(* Logix 5000 project; controller GEA_Test_Chamber vendor 1 type 14 code 196 rev 32.14; software revision 32.04; part 3 of 11 *)
(* tags used below, declared in another part *)
   Inp_Enable : BOOL;
   Ref_Connection : raC_UDT_ModbusServerBase;
   Ref_ModbusData : raC_UDT_ModbusServerData;
   Sts_ActiveConnections : DINT;   // Number of currently active Client connections.
   Ref_MsgDelete : MESSAGE;
   Ref_MsgDeleteAll : MESSAGE;
   Sts_EN : BOOL;
   Sts_Waiting : BOOL;
   Sts_Accepted : BOOL;
   Sts_Faulted : BOOL;
   Sts_LastError : DINT;   // The last recorded socket error for this connection. 0 good, -2- Write Error, -4 - Read Error, -6 connection failed, -7 D
   Wrk_MSGStep : DINT;
   Wrk_BaseInstance : DINT;
   Wrk_WrIndex : DINT;
   Wrk_TransIndex : DINT;
   Wrk_TimerIndex : DINT;
   Wrk_ClrReqIndex : DINT;
   Wrk_AcceptInstance : DINT;
   Wrk_InstSize : DINT;
   Wrk_RdWrIndex : DINT;
   Wrk_TempActConn : DINT;
   Wrk_InstIndex : DINT;
   Wrk_LastInstIndex : DINT;
   Wrk_OkToIncement : BOOL;
   Wrk_StepLockTimer : TIMER;
   Wrk_TempTime : DINT;
   Wrk_Instances : raC_UDT_ModbusServerRWSocket[10];
   Wrk_Controller_Type : DINT;
   Wrk_Controller_Name : SINT[33];
   Wrk_InitCompleted : BOOL;
   Wrk_InstIndex2 : DINT;
   Wrk_InstIndex3 : DINT;
   HMI_Tab : DINT;
   wrk_temp_Instances : raC_UDT_ModbusServerRWSocketInfo[10];
   wrk_FAL_Addr : CONTROL;
   wrk_LoopIndex : DINT;
   wrk_AddrIndex : DINT;
   HMI : raC_UDT_ModbusServerHMI;
   wrk_FAL_01 : CONTROL;
(* raC_Opr_NetModbusTCPServer, continued *)

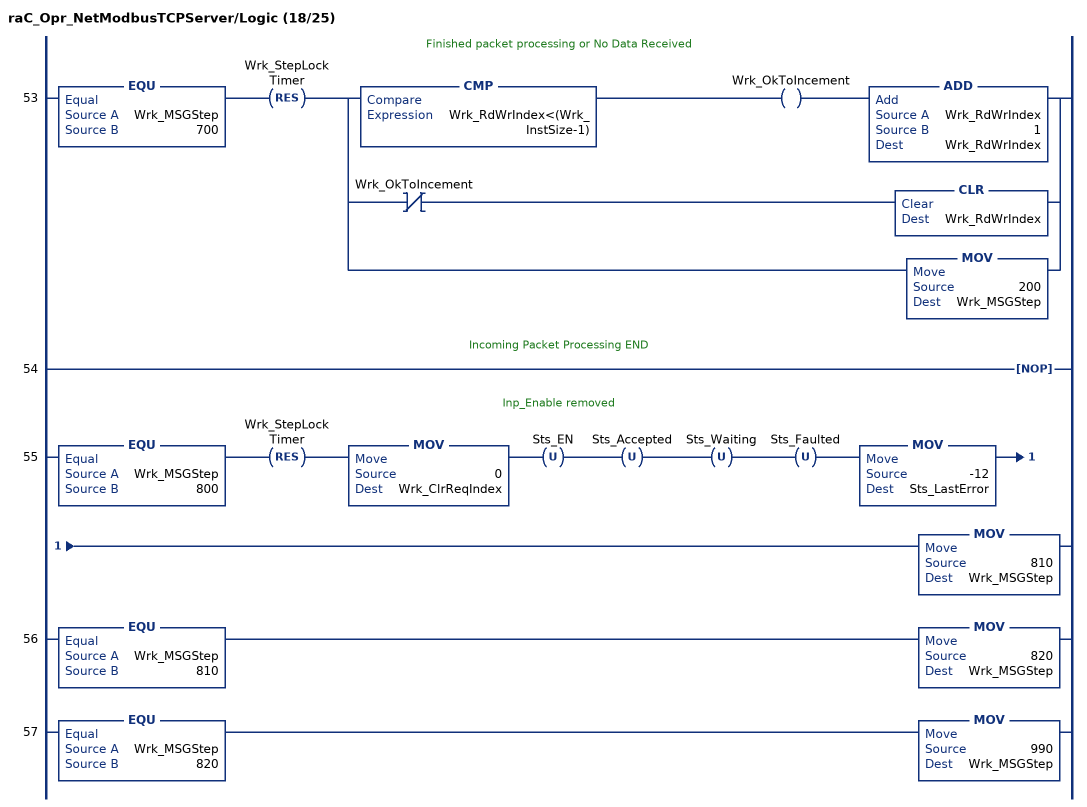
   // Finished packet processing or No Data Received
   53: EQU(Wrk_MSGStep,700)RES(Wrk_StepLockTimer)[CMP(Wrk_RdWrIndex<(Wrk_InstSize-1)) OTE(Wrk_OkToIncement) ADD(Wrk_RdWrIndex,1,Wrk_RdWrIndex) ,XIO(Wrk_OkToIncement) CLR(Wrk_RdWrIndex) ,MOV(200,Wrk_MSGStep) ];
   // Incoming Packet Processing END
   54: NOP();
   // Inp_Enable removed
   55: EQU(Wrk_MSGStep,800)RES(Wrk_StepLockTimer)MOV(0,Wrk_ClrReqIndex)OTU(Sts_EN)OTU(Sts_Accepted)OTU(Sts_Waiting)OTU(Sts_Faulted)MOV(-12,Sts_LastError)MOV(810,Wrk_MSGStep);
   56: EQU(Wrk_MSGStep,810)MOV(820,Wrk_MSGStep);
   57: EQU(Wrk_MSGStep,820)MOV(990,Wrk_MSGStep);
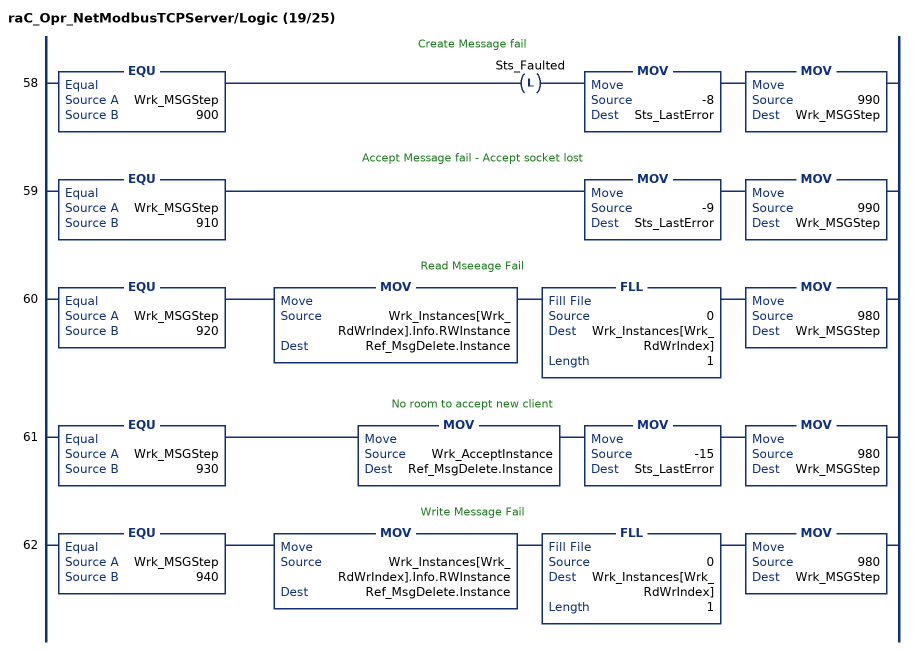
   // Create Message fail
   58: EQU(Wrk_MSGStep,900)OTL(Sts_Faulted)MOV(-8,Sts_LastError)MOV(990,Wrk_MSGStep);
   // Accept Message fail - Accept socket lost
   59: EQU(Wrk_MSGStep,910)MOV(-9,Sts_LastError)MOV(990,Wrk_MSGStep);
   // Read Mseeage Fail
   60: EQU(Wrk_MSGStep,920)MOV(Wrk_Instances[Wrk_RdWrIndex].Info.RWInstance,Ref_MsgDelete.Instance)FLL(0,Wrk_Instances[Wrk_RdWrIndex],1)MOV(980,Wrk_MSGStep);
   // No room to accept new client
   61: EQU(Wrk_MSGStep,930)MOV(Wrk_AcceptInstance,Ref_MsgDelete.Instance)MOV(-15,Sts_LastError)MOV(980,Wrk_MSGStep);
   // Write Message Fail
   62: EQU(Wrk_MSGStep,940)MOV(Wrk_Instances[Wrk_RdWrIndex].Info.RWInstance,Ref_MsgDelete.Instance)FLL(0,Wrk_Instances[Wrk_RdWrIndex],1)MOV(980,Wrk_MSGStep);
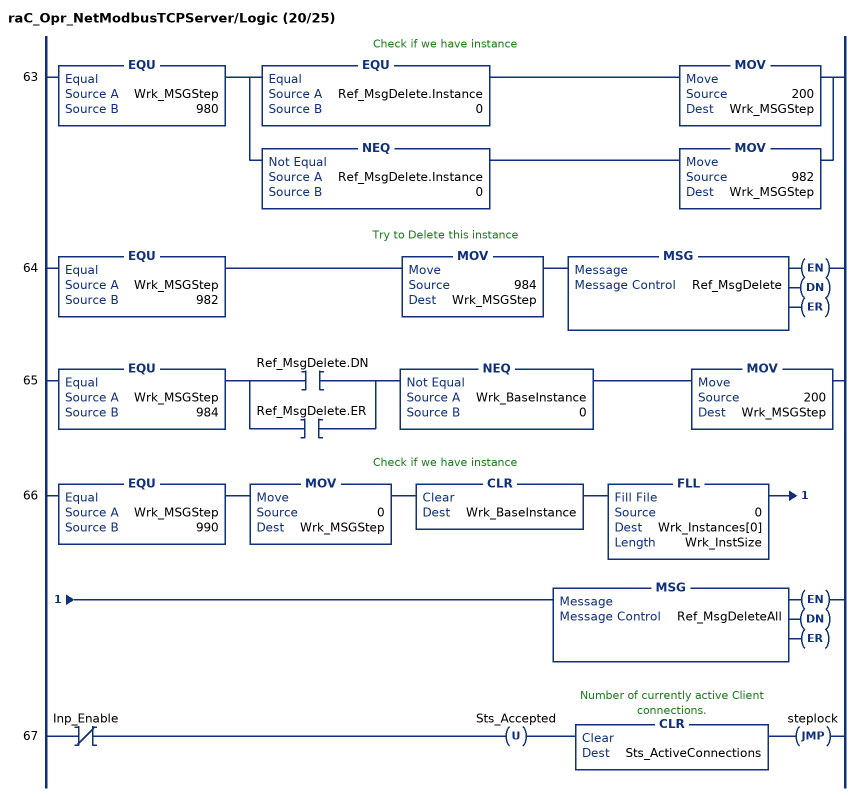
   // Check if we have instance
   63: EQU(Wrk_MSGStep,980)[EQU(Ref_MsgDelete.Instance,0) MOV(200,Wrk_MSGStep) ,NEQ(Ref_MsgDelete.Instance,0) MOV(982,Wrk_MSGStep) ];
   // Try to Delete this instance
   64: EQU(Wrk_MSGStep,982)MOV(984,Wrk_MSGStep)MSG(Ref_MsgDelete);
   65: EQU(Wrk_MSGStep,984)[XIC(Ref_MsgDelete.DN) ,XIC(Ref_MsgDelete.ER) ]NEQ(Wrk_BaseInstance,0)MOV(200,Wrk_MSGStep);
   // Check if we have instance
   66: EQU(Wrk_MSGStep,990)MOV(0,Wrk_MSGStep)CLR(Wrk_BaseInstance)FLL(0,Wrk_Instances[0],Wrk_InstSize)MSG(Ref_MsgDeleteAll);
   67: XIO(Inp_Enable)OTU(Sts_Accepted)CLR(Sts_ActiveConnections)JMP(steplock);
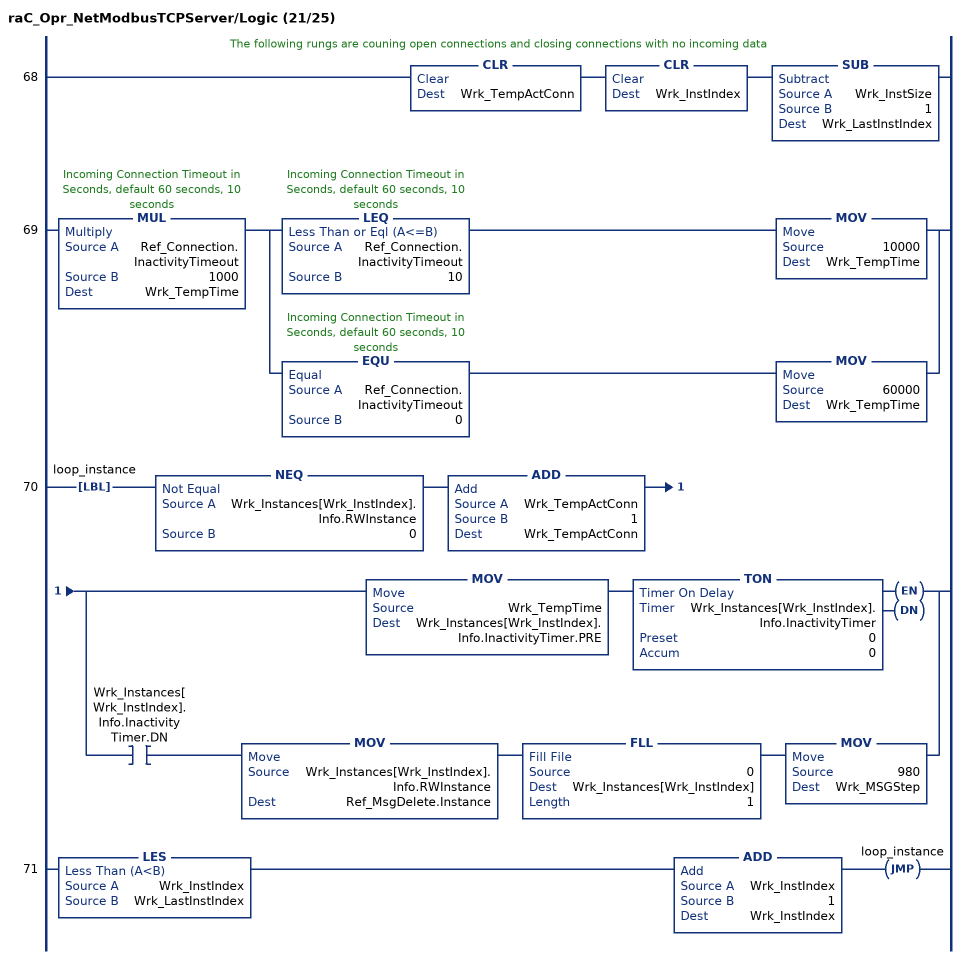
   // The following rungs are couning open connections and closing connections with no incoming data
   68: CLR(Wrk_TempActConn)CLR(Wrk_InstIndex)SUB(Wrk_InstSize,1,Wrk_LastInstIndex);
   69: MUL(Ref_Connection.InactivityTimeout,1000,Wrk_TempTime)[LEQ(Ref_Connection.InactivityTimeout,10) MOV(10000,Wrk_TempTime) ,EQU(Ref_Connection.InactivityTimeout,0) MOV(60000,Wrk_TempTime) ];
   70: LBL(loop_instance)NEQ(Wrk_Instances[Wrk_InstIndex].Info.RWInstance,0)ADD(Wrk_TempActConn,1,Wrk_TempActConn)[MOV(Wrk_TempTime,Wrk_Instances[Wrk_InstIndex].Info.InactivityTimer.PRE) TON(Wrk_Instances[Wrk_InstIndex].Info.InactivityTimer,0,0) ,XIC(Wrk_Instances[Wrk_InstIndex].Info.InactivityTimer.DN) MOV(Wrk_Instances[Wrk_InstIndex].Info.RWInstance,Ref_MsgDelete.Instance) FLL(0,Wrk_Instances[Wrk_InstIndex],1) MOV(980,Wrk_MSGStep) ];
   71: LES(Wrk_InstIndex,Wrk_LastInstIndex)ADD(Wrk_InstIndex,1,Wrk_InstIndex)JMP(loop_instance);
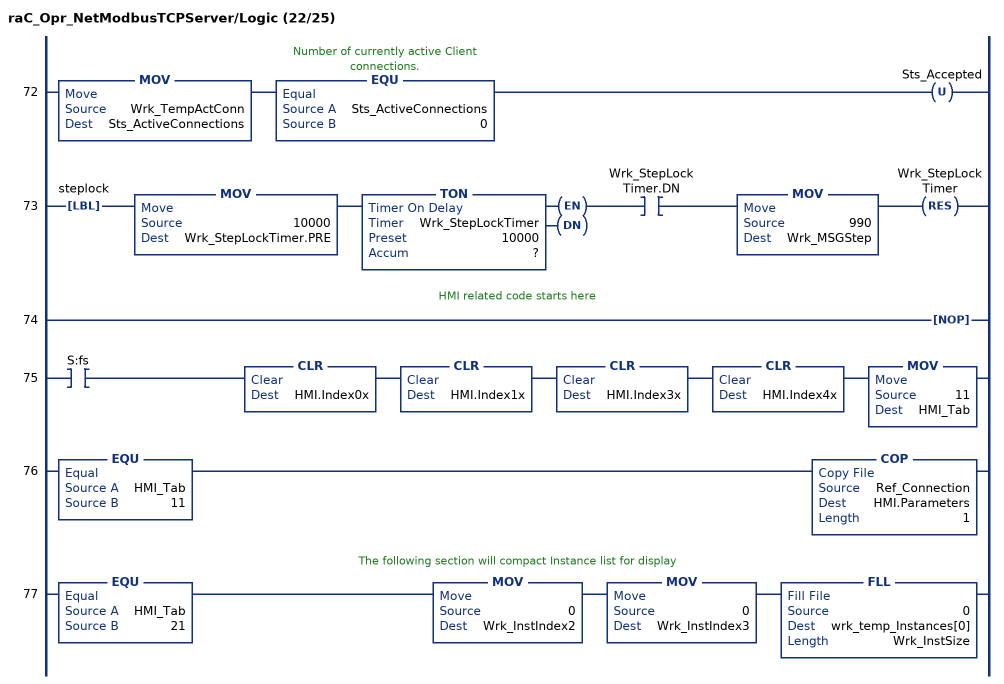
   72: MOV(Wrk_TempActConn,Sts_ActiveConnections)EQU(Sts_ActiveConnections,0)OTU(Sts_Accepted);
   73: LBL(steplock)MOV(10000,Wrk_StepLockTimer.PRE)TON(Wrk_StepLockTimer,?,?)XIC(Wrk_StepLockTimer.DN)MOV(990,Wrk_MSGStep)RES(Wrk_StepLockTimer);
   // HMI related code starts here
   74: NOP();
   75: XIC(S:fs)CLR(HMI.Index0x)CLR(HMI.Index1x)CLR(HMI.Index3x)CLR(HMI.Index4x)MOV(11,HMI_Tab);
   76: EQU(HMI_Tab,11)COP(Ref_Connection,HMI.Parameters,1);
   // The following section will compact Instance list for display
   77: EQU(HMI_Tab,21)MOV(0,Wrk_InstIndex2)MOV(0,Wrk_InstIndex3)FLL(0,wrk_temp_Instances[0],Wrk_InstSize);
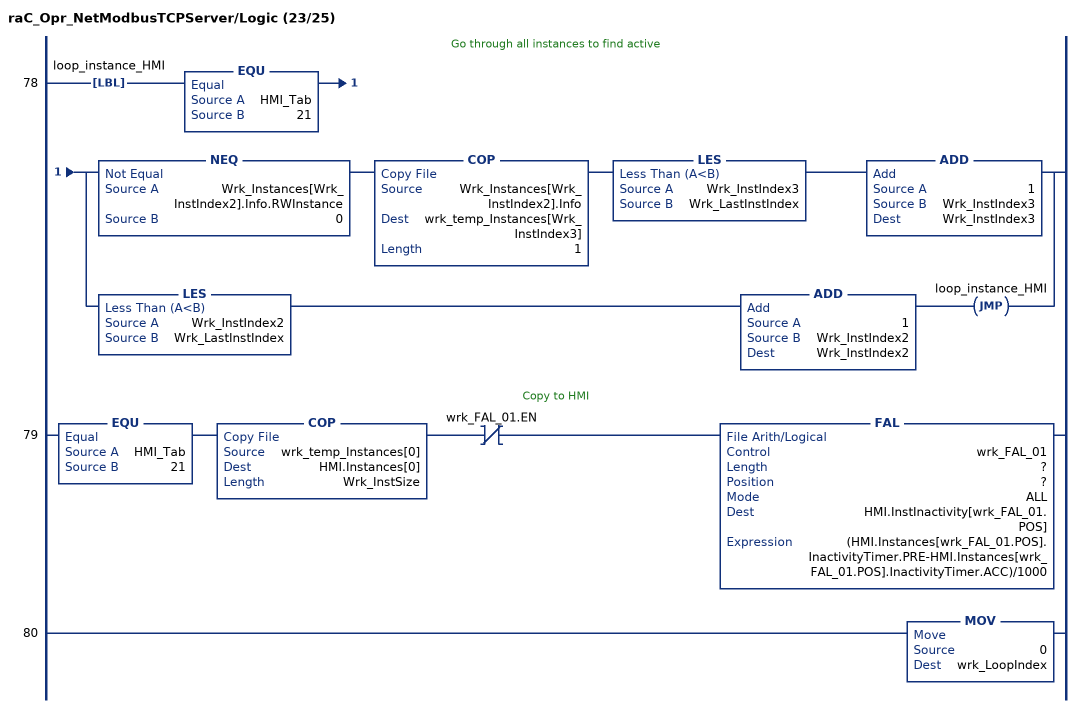
   // Go through all instances to find active
   78: LBL(loop_instance_HMI)EQU(HMI_Tab,21)[NEQ(Wrk_Instances[Wrk_InstIndex2].Info.RWInstance,0) COP(Wrk_Instances[Wrk_InstIndex2].Info,wrk_temp_Instances[Wrk_InstIndex3],1) LES(Wrk_InstIndex3,Wrk_LastInstIndex) ADD(1,Wrk_InstIndex3,Wrk_InstIndex3) ,LES(Wrk_InstIndex2,Wrk_LastInstIndex) ADD(1,Wrk_InstIndex2,Wrk_InstIndex2) JMP(loop_instance_HMI) ];
   // Copy to HMI
   79: EQU(HMI_Tab,21)COP(wrk_temp_Instances[0],HMI.Instances[0],Wrk_InstSize)XIO(wrk_FAL_01.EN)FAL(wrk_FAL_01,?,?,ALL,HMI.InstInactivity[wrk_FAL_01.POS],(HMI.Instances[wrk_FAL_01.POS].InactivityTimer.PRE-HMI.Instances[wrk_FAL_01.POS].InactivityTimer.ACC)/1000);
   80: MOV(0,wrk_LoopIndex);
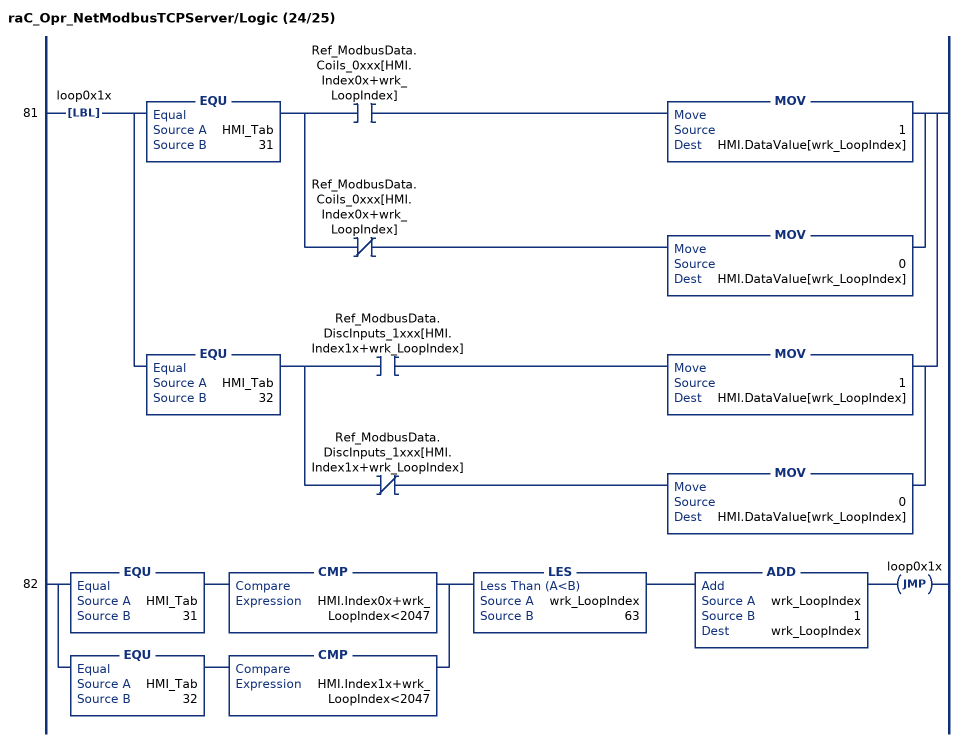
   81: LBL(loop0x1x)[EQU(HMI_Tab,31) [XIC(Ref_ModbusData.Coils_0xxx[HMI.Index0x+wrk_LoopIndex]) MOV(1,HMI.DataValue[wrk_LoopIndex]) ,XIO(Ref_ModbusData.Coils_0xxx[HMI.Index0x+wrk_LoopIndex]) MOV(0,HMI.DataValue[wrk_LoopIndex]) ] ,EQU(HMI_Tab,32) [XIC(Ref_ModbusData.DiscInputs_1xxx[HMI.Index1x+wrk_LoopIndex]) MOV(1,HMI.DataValue[wrk_LoopIndex]) ,XIO(Ref_ModbusData.DiscInputs_1xxx[HMI.Index1x+wrk_LoopIndex]) MOV(0,HMI.DataValue[wrk_LoopIndex]) ] ];
   82: [EQU(HMI_Tab,31) CMP(HMI.Index0x+wrk_LoopIndex<2047) ,EQU(HMI_Tab,32) CMP(HMI.Index1x+wrk_LoopIndex<2047) ]LES(wrk_LoopIndex,63)ADD(wrk_LoopIndex,1,wrk_LoopIndex)JMP(loop0x1x);
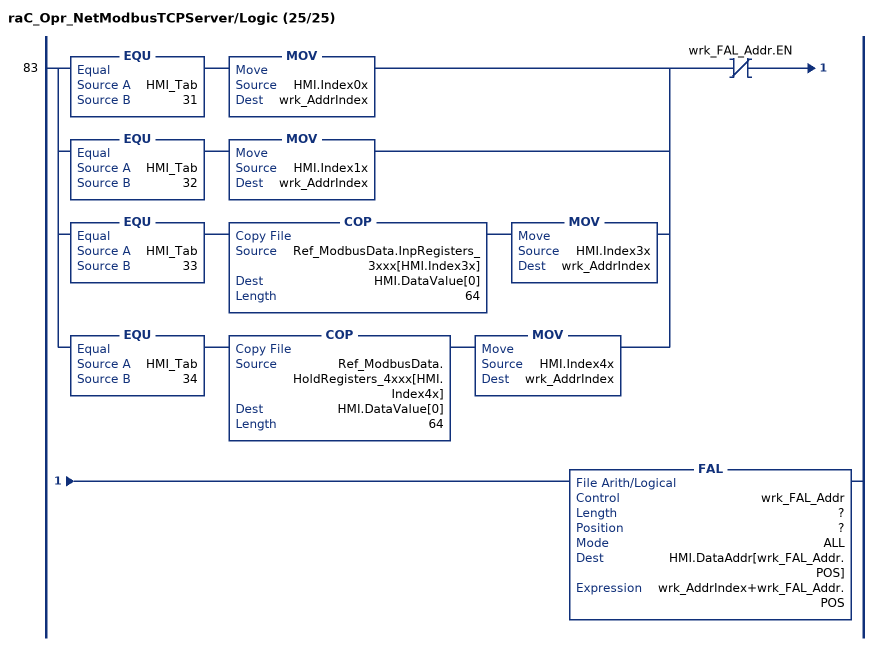
   83: [EQU(HMI_Tab,31) MOV(HMI.Index0x,wrk_AddrIndex) ,EQU(HMI_Tab,32) MOV(HMI.Index1x,wrk_AddrIndex) ,EQU(HMI_Tab,33) COP(Ref_ModbusData.InpRegisters_3xxx[HMI.Index3x],HMI.DataValue[0],64) MOV(HMI.Index3x,wrk_AddrIndex) ,EQU(HMI_Tab,34) COP(Ref_ModbusData.HoldRegisters_4xxx[HMI.Index4x],HMI.DataValue[0],64) MOV(HMI.Index4x,wrk_AddrIndex) ]XIO(wrk_FAL_Addr.EN)FAL(wrk_FAL_Addr,?,?,ALL,HMI.DataAddr[wrk_FAL_Addr.POS],wrk_AddrIndex+wrk_FAL_Addr.POS);
END_ROUTINE

ROUTINE Prescan   (* ladder *)
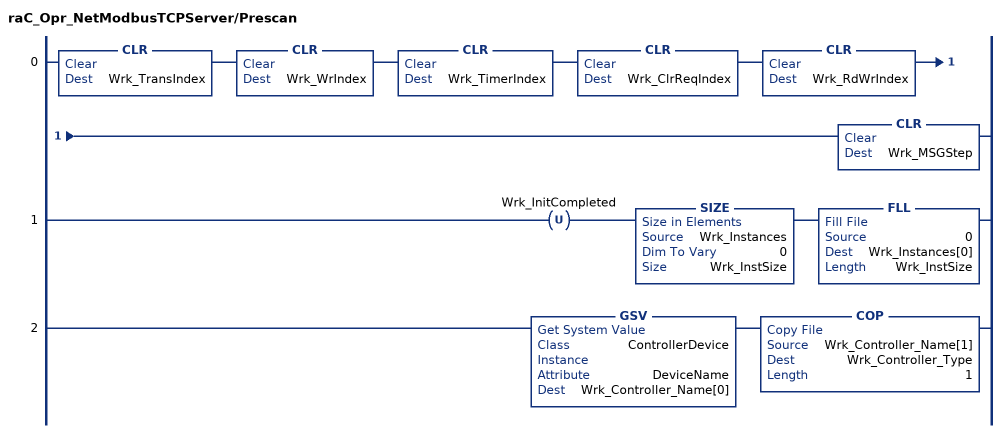
   0: CLR(Wrk_TransIndex)CLR(Wrk_WrIndex)CLR(Wrk_TimerIndex)CLR(Wrk_ClrReqIndex)CLR(Wrk_RdWrIndex)CLR(Wrk_MSGStep);
   1: OTU(Wrk_InitCompleted)SIZE(Wrk_Instances,0,Wrk_InstSize)FLL(0,Wrk_Instances[0],Wrk_InstSize);
   2: GSV(ControllerDevice,,DeviceName,Wrk_Controller_Name[0])COP(Wrk_Controller_Name[1],Wrk_Controller_Type,1);
END_ROUTINE
END_ADD_ON_INSTRUCTION

ADD_ON_INSTRUCTION raC_Tec_NetModbusTCPClient_BuildReqStr   (* revision 2.1, ExecutePrescan *)
// This routine builds a request string.
// Revision note:
// Moved to DINT in BeginAddress with boundary enforcement
VAR_IN_OUT
   Transaction : raC_UDT_ModbusClientTransaction; {required}
   ModbusData : raC_UDT_ModbusClientData; {required}
END_VAR
VAR_OUTPUT
   ER : BOOL; {access Read Only, visible}
END_VAR
VAR
   Wrk_TempInt : INT; {access None}
   Wrk_TempBeginInt : INT; {access None}
   Wrk_TempASCII_462 : STR0462; {access None}
   Wrk_Bit : DINT; {access None}
   Wrk_Byte : DINT; {access None}
   Wrk_Index : DINT; {access None}
   Wrk_LastAddr : DINT; {access None}
   Wrk_ValidRemoteRange : BOOL; {access None}
END_VAR

ROUTINE Logic   (* ladder *)
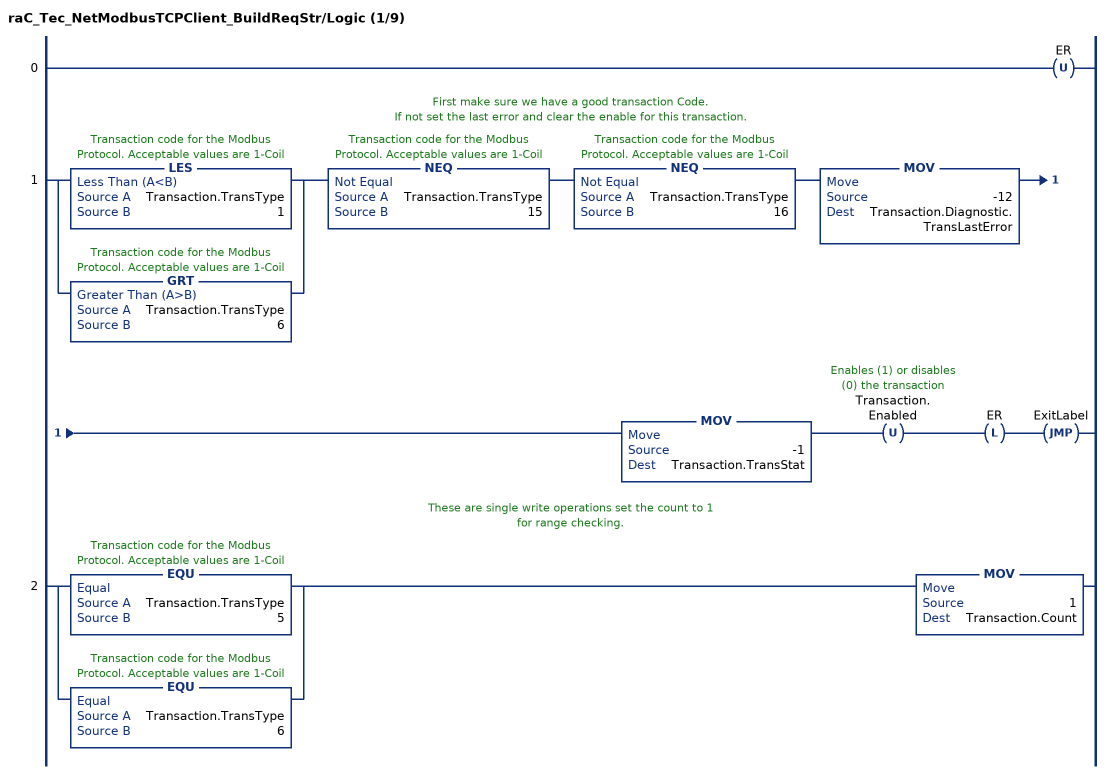
   0: OTU(ER);
   // First make sure we have a good transaction Code.
   // If not set the last error and clear the enable for this transaction.
   1: [LES(Transaction.TransType,1) ,GRT(Transaction.TransType,6) ]NEQ(Transaction.TransType,15)NEQ(Transaction.TransType,16)MOV(-12,Transaction.Diagnostic.TransLastError)MOV(-1,Transaction.TransStat)OTU(Transaction.Enabled)OTL(ER)JMP(ExitLabel);
   // These are single write operations set the count to 1
   //  for range checking.
   2: [EQU(Transaction.TransType,5) ,EQU(Transaction.TransType,6) ]MOV(1,Transaction.Count);
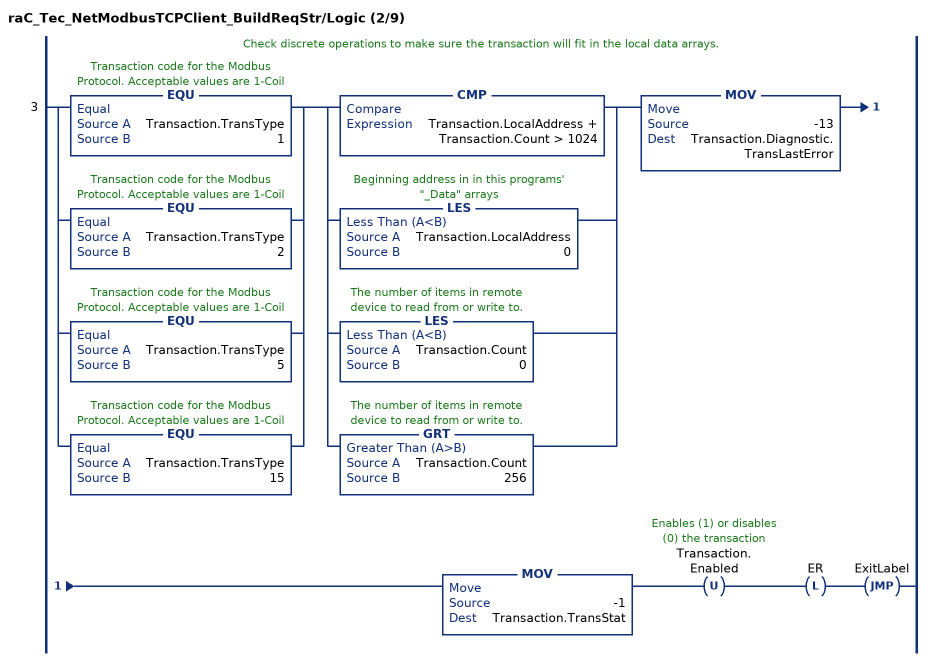
   // Check discrete operations to make sure the transaction will fit in the local data arrays.
   3: [EQU(Transaction.TransType,1) ,EQU(Transaction.TransType,2) ,EQU(Transaction.TransType,5) ,EQU(Transaction.TransType,15) ][CMP(Transaction.LocalAddress + Transaction.Count > 1024) ,LES(Transaction.LocalAddress,0) ,LES(Transaction.Count,0) ,GRT(Transaction.Count,256) ]MOV(-13,Transaction.Diagnostic.TransLastError)MOV(-1,Transaction.TransStat)OTU(Transaction.Enabled)OTL(ER)JMP(ExitLabel);
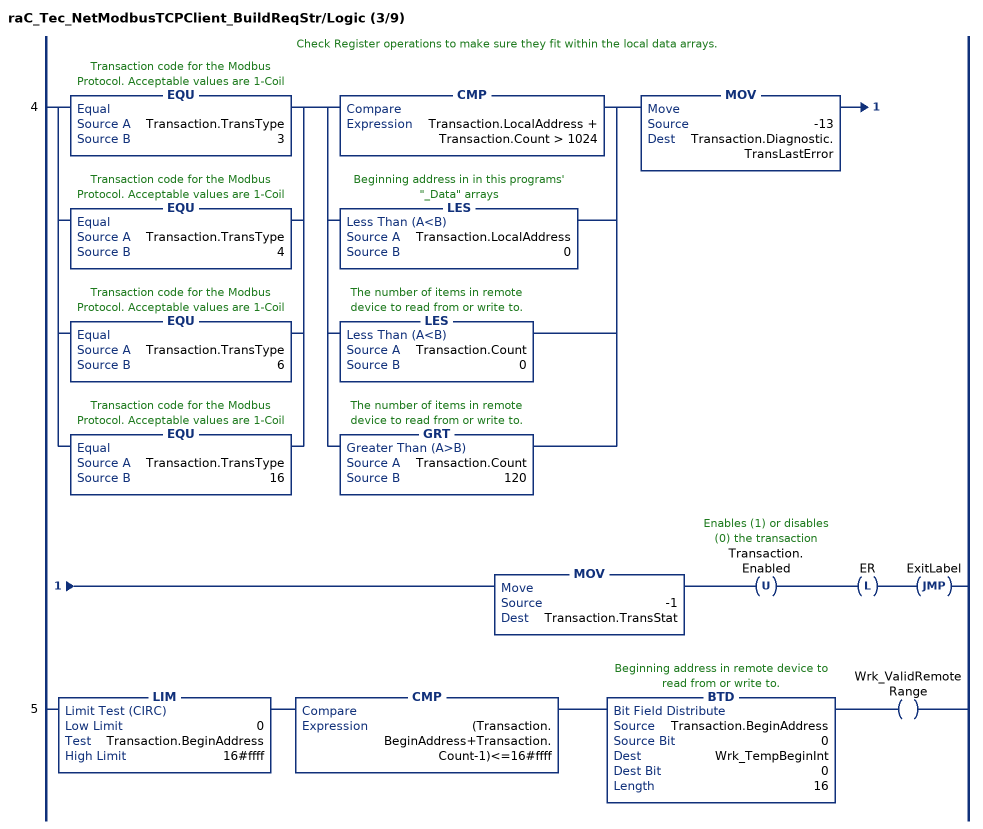
   // Check Register operations to make sure they fit within the local data arrays.
   4: [EQU(Transaction.TransType,3) ,EQU(Transaction.TransType,4) ,EQU(Transaction.TransType,6) ,EQU(Transaction.TransType,16) ][CMP(Transaction.LocalAddress + Transaction.Count > 1024) ,LES(Transaction.LocalAddress,0) ,LES(Transaction.Count,0) ,GRT(Transaction.Count,120) ]MOV(-13,Transaction.Diagnostic.TransLastError)MOV(-1,Transaction.TransStat)OTU(Transaction.Enabled)OTL(ER)JMP(ExitLabel);
   5: LIM(0,Transaction.BeginAddress,16#ffff)CMP((Transaction.BeginAddress+Transaction.Count-1)<=16#ffff)BTD(Transaction.BeginAddress,0,Wrk_TempBeginInt,0,16)OTE(Wrk_ValidRemoteRange);
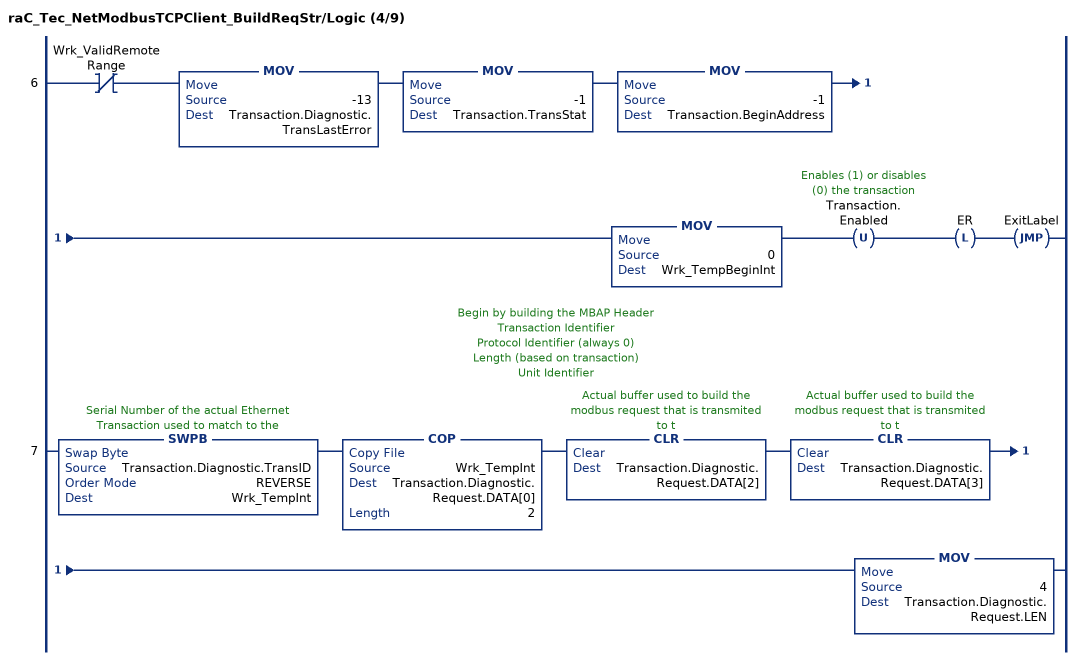
   6: XIO(Wrk_ValidRemoteRange)MOV(-13,Transaction.Diagnostic.TransLastError)MOV(-1,Transaction.TransStat)MOV(-1,Transaction.BeginAddress)MOV(0,Wrk_TempBeginInt)OTU(Transaction.Enabled)OTL(ER)JMP(ExitLabel);
   // Begin by building the MBAP Header
   // Transaction Identifier
   // Protocol Identifier (always 0)
   // Length (based on transaction)
   // Unit Identifier
   7: SWPB(Transaction.Diagnostic.TransID,REVERSE,Wrk_TempInt)COP(Wrk_TempInt,Transaction.Diagnostic.Request.DATA[0],2)CLR(Transaction.Diagnostic.Request.DATA[2])CLR(Transaction.Diagnostic.Request.DATA[3])MOV(4,Transaction.Diagnostic.Request.LEN);
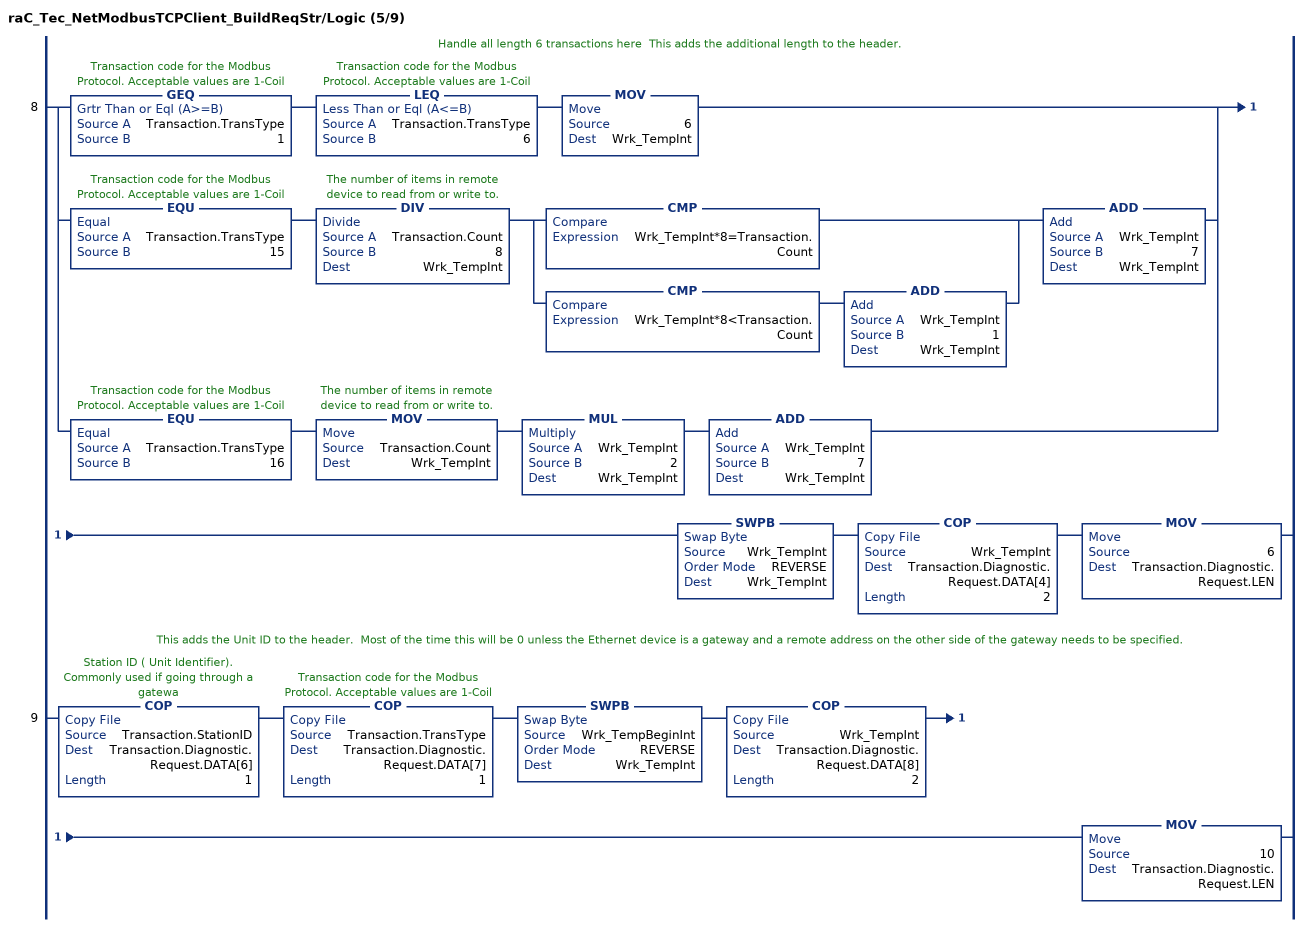
   // Handle all length 6 transactions here  This adds the additional length to the header.
   8: [GEQ(Transaction.TransType,1) LEQ(Transaction.TransType,6) MOV(6,Wrk_TempInt) ,EQU(Transaction.TransType,15) DIV(Transaction.Count,8,Wrk_TempInt) [CMP(Wrk_TempInt*8=Transaction.Count) ,CMP(Wrk_TempInt*8<Transaction.Count) ADD(Wrk_TempInt,1,Wrk_TempInt) ] ADD(Wrk_TempInt,7,Wrk_TempInt) ,EQU(Transaction.TransType,16) MOV(Transaction.Count,Wrk_TempInt) MUL(Wrk_TempInt,2,Wrk_TempInt) ADD(Wrk_TempInt,7,Wrk_TempInt) ]SWPB(Wrk_TempInt,REVERSE,Wrk_TempInt)COP(Wrk_TempInt,Transaction.Diagnostic.Request.DATA[4],2)MOV(6,Transaction.Diagnostic.Request.LEN);
   // This adds the Unit ID to the header.  Most of the time this will be 0 unless the Ethernet device is a gateway and a remote address on the other side of the gateway needs to be specified.
   9: COP(Transaction.StationID,Transaction.Diagnostic.Request.DATA[6],1)COP(Transaction.TransType,Transaction.Diagnostic.Request.DATA[7],1)SWPB(Wrk_TempBeginInt,REVERSE,Wrk_TempInt)COP(Wrk_TempInt,Transaction.Diagnostic.Request.DATA[8],2)MOV(10,Transaction.Diagnostic.Request.LEN);
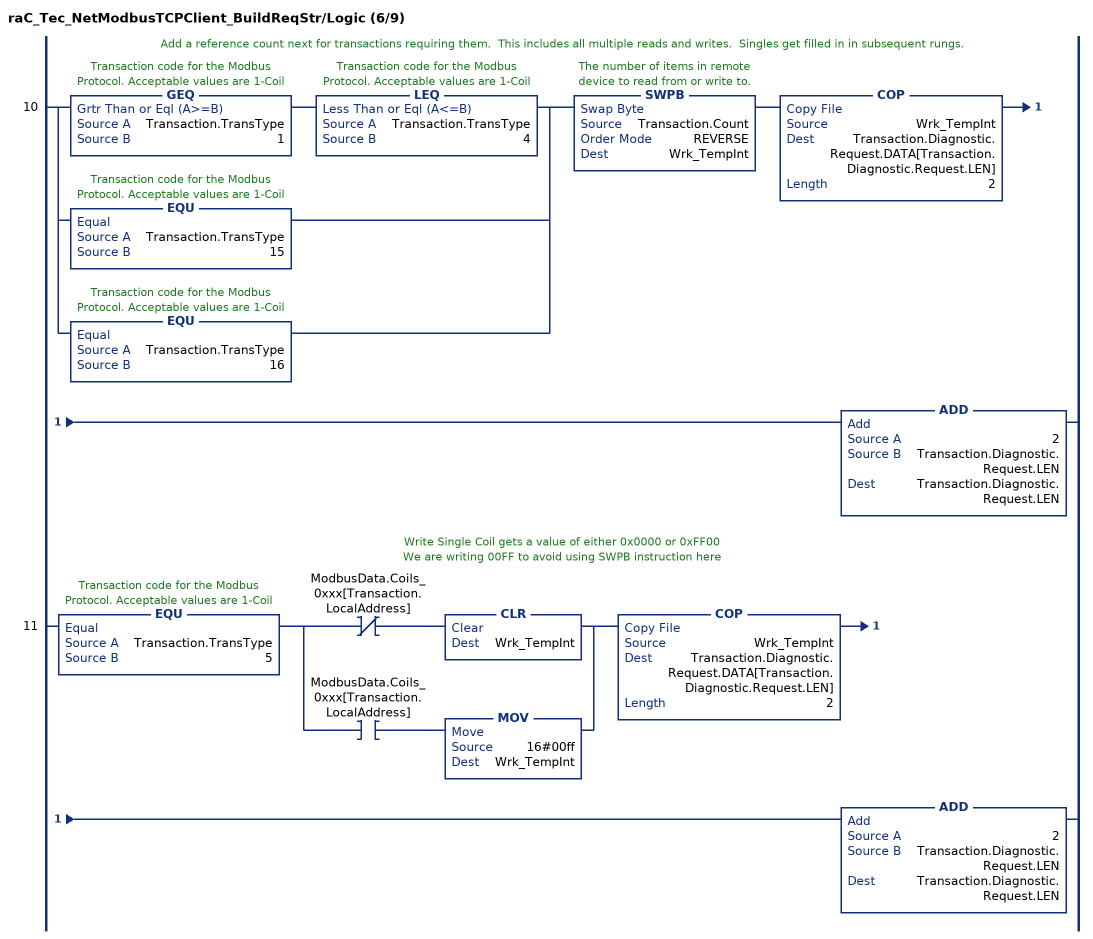
   // Add a reference count next for transactions requiring them.  This includes all multiple reads and writes.  Singles get filled in in subsequent rungs.
   10: [GEQ(Transaction.TransType,1) LEQ(Transaction.TransType,4) ,EQU(Transaction.TransType,15) ,EQU(Transaction.TransType,16) ]SWPB(Transaction.Count,REVERSE,Wrk_TempInt)COP(Wrk_TempInt,Transaction.Diagnostic.Request.DATA[Transaction.Diagnostic.Request.LEN],2)ADD(2,Transaction.Diagnostic.Request.LEN,Transaction.Diagnostic.Request.LEN);
   // Write Single Coil gets a value of either 0x0000 or 0xFF00
   // We are writing 00FF to avoid using SWPB instruction here
   11: EQU(Transaction.TransType,5)[XIO(ModbusData.Coils_0xxx[Transaction.LocalAddress]) CLR(Wrk_TempInt) ,XIC(ModbusData.Coils_0xxx[Transaction.LocalAddress]) MOV(16#00ff,Wrk_TempInt) ]COP(Wrk_TempInt,Transaction.Diagnostic.Request.DATA[Transaction.Diagnostic.Request.LEN],2)ADD(2,Transaction.Diagnostic.Request.LEN,Transaction.Diagnostic.Request.LEN);
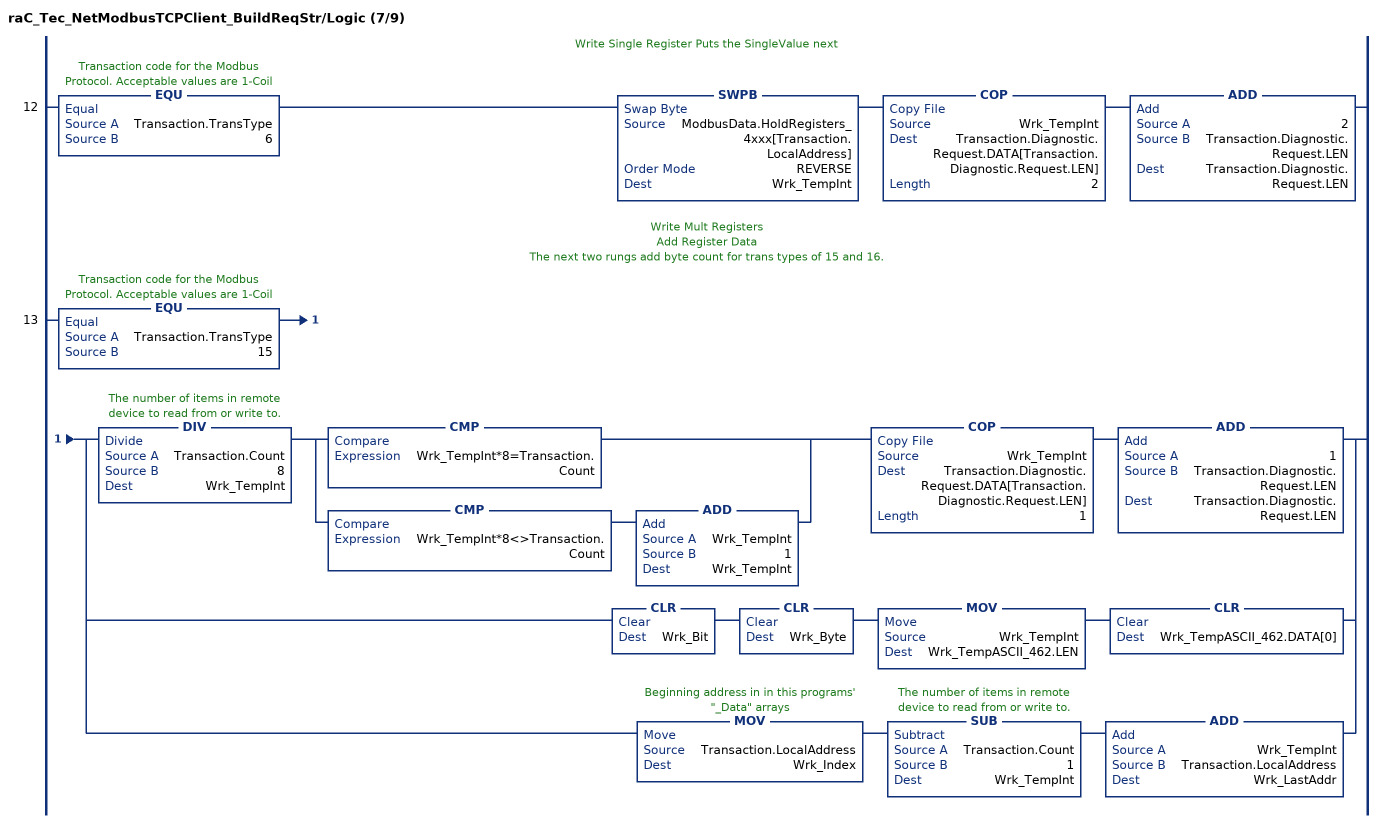
   // Write Single Register Puts the SingleValue next
   12: EQU(Transaction.TransType,6)SWPB(ModbusData.HoldRegisters_4xxx[Transaction.LocalAddress],REVERSE,Wrk_TempInt)COP(Wrk_TempInt,Transaction.Diagnostic.Request.DATA[Transaction.Diagnostic.Request.LEN],2)ADD(2,Transaction.Diagnostic.Request.LEN,Transaction.Diagnostic.Request.LEN);
   // Write Mult Registers
   // Add Register Data
   // The next two rungs add byte count for trans types of 15 and 16.
   13: EQU(Transaction.TransType,15)[DIV(Transaction.Count,8,Wrk_TempInt) [CMP(Wrk_TempInt*8=Transaction.Count) ,CMP(Wrk_TempInt*8<>Transaction.Count) ADD(Wrk_TempInt,1,Wrk_TempInt) ] COP(Wrk_TempInt,Transaction.Diagnostic.Request.DATA[Transaction.Diagnostic.Request.LEN],1) ADD(1,Transaction.Diagnostic.Request.LEN,Transaction.Diagnostic.Request.LEN) ,CLR(Wrk_Bit) CLR(Wrk_Byte) MOV(Wrk_TempInt,Wrk_TempASCII_462.LEN) CLR(Wrk_TempASCII_462.DATA[0]) ,MOV(Transaction.LocalAddress,Wrk_Index) SUB(Transaction.Count,1,Wrk_TempInt) ADD(Wrk_TempInt,Transaction.LocalAddress,Wrk_LastAddr) ];
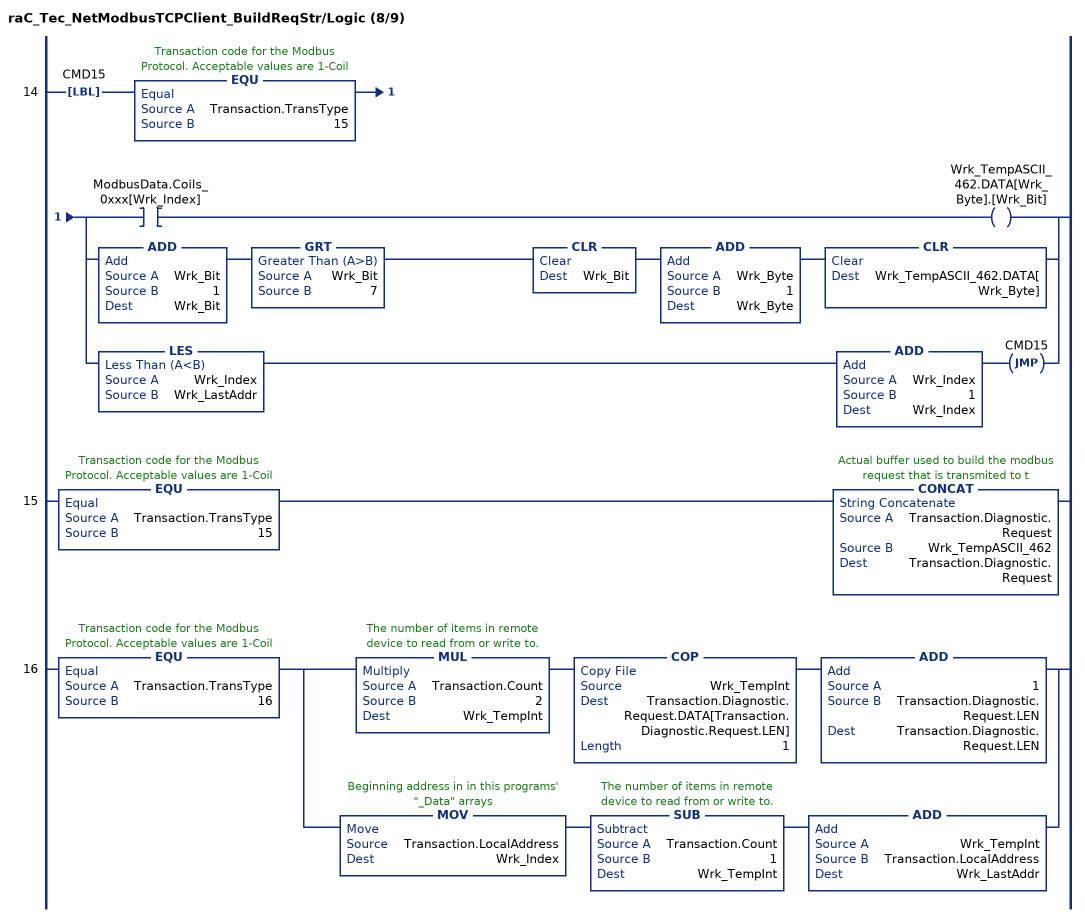
   14: LBL(CMD15)EQU(Transaction.TransType,15)[XIC(ModbusData.Coils_0xxx[Wrk_Index]) OTE(Wrk_TempASCII_462.DATA[Wrk_Byte].[Wrk_Bit]) ,ADD(Wrk_Bit,1,Wrk_Bit) GRT(Wrk_Bit,7) CLR(Wrk_Bit) ADD(Wrk_Byte,1,Wrk_Byte) CLR(Wrk_TempASCII_462.DATA[Wrk_Byte]) ,LES(Wrk_Index,Wrk_LastAddr) ADD(Wrk_Index,1,Wrk_Index) JMP(CMD15) ];
   15: EQU(Transaction.TransType,15)CONCAT(Transaction.Diagnostic.Request,Wrk_TempASCII_462,Transaction.Diagnostic.Request);
   16: EQU(Transaction.TransType,16)[MUL(Transaction.Count,2,Wrk_TempInt) COP(Wrk_TempInt,Transaction.Diagnostic.Request.DATA[Transaction.Diagnostic.Request.LEN],1) ADD(1,Transaction.Diagnostic.Request.LEN,Transaction.Diagnostic.Request.LEN) ,MOV(Transaction.LocalAddress,Wrk_Index) SUB(Transaction.Count,1,Wrk_TempInt) ADD(Wrk_TempInt,Transaction.LocalAddress,Wrk_LastAddr) ];
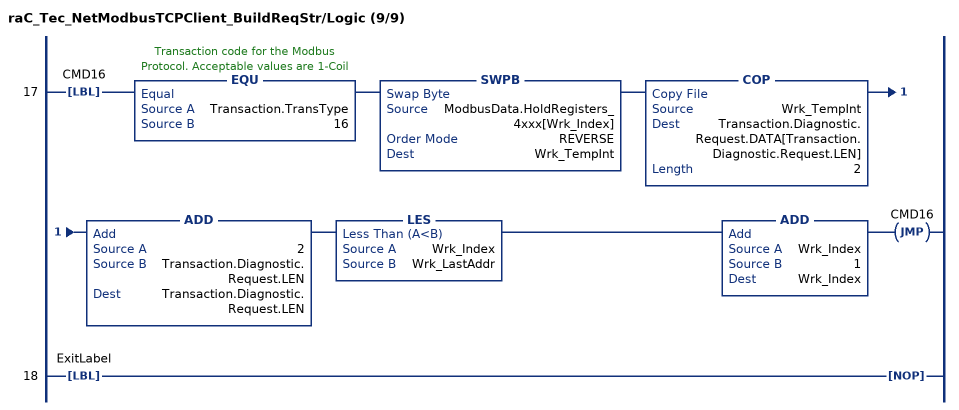
   17: LBL(CMD16)EQU(Transaction.TransType,16)SWPB(ModbusData.HoldRegisters_4xxx[Wrk_Index],REVERSE,Wrk_TempInt)COP(Wrk_TempInt,Transaction.Diagnostic.Request.DATA[Transaction.Diagnostic.Request.LEN],2)ADD(2,Transaction.Diagnostic.Request.LEN,Transaction.Diagnostic.Request.LEN)LES(Wrk_Index,Wrk_LastAddr)ADD(Wrk_Index,1,Wrk_Index)JMP(CMD16);
   18: LBL(ExitLabel)NOP();
END_ROUTINE
